FUNCTION_BLOCK AxisRelTestSuite 
VAR
	StubAxis : AXIS_REF;
	iStubTask : I_Task;
	TestAxisRel : MoveRelTask := (AxisRef := stubaxis);
	TestObjRunner : ObjectRunner<99>;
	ObjTestSuite : TestSuite<TestSuiteParameter.MaxTestCount>(ResultFile := JUnitResultFile) := (TestSuiteName := 'Object Test Suite');
END_VAR

CheckCorrectRegistration_Test();
TaskAcceptValidCommand_Test();
TaskRejectsZeroVeloCommand_Test();

METHOD CheckCorrectRegistration_Test : BOOL
VAR_INST
	Expected : BOOL := TRUE;
	Actual	 : bool;
END_VAR
IF ObjTestSuite.Test(__POUNAME()).ExecuteTest() THEN
	TestAxisRel.RegisterWithParent(TestObjRunner);
	Actual := TestObjRunner.CyclicModuleCount = TestObjRunner.AbortableModuleCount AND
				TestObjRunner.CyclicModuleCount = TestObjRunner.TaskModuleCount;
	ObjTestSuite.Test(__POUNAME()).AssertEqual(Expected, Actual);
END_IF
END_METHOD

METHOD TaskAcceptValidCommand_Test : BOOL
VAR_INST
	Expected : BOOL := TRUE;
	Actual	 : bool;
END_VAR
IF ObjTestSuite.Test(__POUNAME()).ExecuteTest() THEN
	Actual := SUCCEEDED(TestAxisRel.MoveBy(100.0, 300.0));
	TestAxisRel.Abort();
	ObjTestSuite.Test(__POUNAME()).AssertEqual(Expected, Actual);
END_IF
END_METHOD

METHOD TaskRejectsZeroVeloCommand_Test : BOOL
VAR_INST
	Expected : BOOL := TRUE;
	Actual	 : bool;
END_VAR
IF ObjTestSuite.Test(__POUNAME()).ExecuteTest() THEN
	Actual := FAILED(TestAxisRel.MoveBy(100.0, 0.0));
	TestAxisRel.Abort();
	ObjTestSuite.Test(__POUNAME()).AssertEqual(Expected, Actual);
END_IF
END_METHOD

END_FUNCTION_BLOCK

(* stored: Version 1.1.0.1
   POU AxisRelTestSuite: Id {17fb2fd6-f573-4d0a-9afb-f84bca683c76}, SpecialFunc None
   Method CheckCorrectRegistration_Test: Id {0e1e6947-5948-4ff9-97fd-75c449021a2d}
   Method TaskAcceptValidCommand_Test: Id {b41aa70b-a86c-411e-a753-699b9539763a}
   Method TaskRejectsZeroVeloCommand_Test: Id {dee3319b-7afd-4544-bf1c-04cd9756e264} *)
